LIN {X 0,Y 44.352,Z 475.064,A -85,B 0,C 180,E1 -30779.969,E2 -30779.969} C_VEL
LIN {X 0,Y 35.444,Z 475.32,A -85,B 0,C 180,E1 -30787.589,E2 -30787.589} C_VEL
LIN {X 0,Y 29.276,Z 474.961,A -85,B 0,C 180,E1 -30796.255,E2 -30796.255} C_VEL
LIN {X 0,Y 22.466,Z 473.712,A -85,B 0,C 180,E1 -30814.655,E2 -30814.655} C_VEL
LIN {X 0,Y 19.51,Z 472.671,A -85,B 0,C 180,E1 -30828.383,E2 -30828.383} C_VEL
LIN {X 0,Y 17,Z 471.328,A -85,B 0,C 180,E1 -30844.896,E2 -30844.896} C_VEL
LIN {X 0,Y 16.61,Z 467.855,A -85,B 0,C 180,E1 -30884.85,E2 -30884.85} C_VEL
LIN {X 0,Y 19.552,Z 465.667,A -85,B 0,C 180,E1 -30899.911,E2 -30899.911} C_VEL
LIN {X 0,Y 20.907,Z 464.867,A -85,B 0,C 180,E1 -30903.377,E2 -30903.377} C_VEL
LIN {X 0,Y 31.045,Z 458.924,A -85,B 0,C 180,E1 -30917.285,E2 -30917.285} C_VEL
LIN {X 0,Y 41.244,Z 451.859,A -85,B 0,C 180,E1 -30924.051,E2 -30924.051} C_VEL
LIN {X 0,Y 51.399,Z 443.285,A -85,B 0,C 180,E1 -30928.242,E2 -30928.242} C_VEL
LIN {X 0,Y 60.425,Z 433.954,A -85,B 0,C 180,E1 -30930.74,E2 -30930.74} C_VEL
LIN {X 0,Y 68.419,Z 423.904,A -85,B 0,C 180,E1 -30932.379,E2 -30932.379} C_VEL
LIN {X 0,Y 75.556,Z 412.822,A -85,B 0,C 180,E1 -30933.554,E2 -30933.554} C_VEL
LIN {X 0,Y 81.798,Z 400.333,A -85,B 0,C 180,E1 -30934.484,E2 -30934.484} C_VEL
LIN {X 0,Y 86.455,Z 387.975,A -85,B 0,C 180,E1 -30935.15,E2 -30935.15} C_VEL
LIN {X 0,Y 89.843,Z 375.107,A -85,B 0,C 180,E1 -30935.553,E2 -30935.553} C_VEL
LIN {X 0,Y 91.232,Z 367.157,A -85,B 0,C 180,E1 -30935.77,E2 -30935.77} C_VEL
LIN {X 0,Y 90.551,Z 364.005,A -85,B 0,C 180,E1 -30939.811,E2 -30939.811} C_VEL
LIN {X 0,Y 90.135,Z 362.029,A -85,B 0,C 180,E1 -30943.737,E2 -30943.737} C_VEL
LIN {X 0,Y 90.077,Z 360.543,A -85,B 0,C 180,E1 -30949.224,E2 -30949.224} C_VEL
LIN {X 0,Y 90.153,Z 360.685,A -85,B 0,C 180,E1 -30951.42,E2 -30951.42} C_VEL
LIN {X 0,Y 90.382,Z 362.249,A -85,B 0,C 180,E1 -30954.99,E2 -30954.99} C_VEL
LIN {X 0,Y 91.055,Z 365.77,A -85,B 0,C 180,E1 -30959.767,E2 -30959.767} C_VEL
LIN {X 0,Y 91.295,Z 367.107,A -85,B 0,C 180,E1 -30961.202,E2 -30961.202} C_VEL
LIN {X 0,Y 89.068,Z 378.985,A -85,B 0,C 180,E1 -30961.537,E2 -30961.537} C_VEL
LIN {X 0,Y 85.544,Z 391.077,A -85,B 0,C 180,E1 -30961.898,E2 -30961.898} C_VEL
LIN {X 0,Y 80.897,Z 402.684,A -85,B 0,C 180,E1 -30962.384,E2 -30962.384} C_VEL
LIN {X 0,Y 74.797,Z 414.427,A -85,B 0,C 180,E1 -30963.235,E2 -30963.235} C_VEL
LIN {X 0,Y 67.835,Z 424.975,A -85,B 0,C 180,E1 -30964.236,E2 -30964.236} C_VEL
LIN {X 0,Y 60.062,Z 434.695,A -85,B 0,C 180,E1 -30965.908,E2 -30965.908} C_VEL
LIN {X 0,Y 51.56,Z 443.447,A -85,B 0,C 180,E1 -30968.156,E2 -30968.156} C_VEL
LIN {X 0,Y 43.026,Z 450.805,A -85,B 0,C 180,E1 -30971.424,E2 -30971.424} C_VEL
LIN {X 0,Y 33.141,Z 457.934,A -85,B 0,C 180,E1 -30977.361,E2 -30977.361} C_VEL
LIN {X 0,Y 23.824,Z 463.593,A -85,B 0,C 180,E1 -30987.718,E2 -30987.718} C_VEL
LIN {X 0,Y 16.117,Z 468.031,A -85,B 0,C 180,E1 -31009.123,E2 -31009.123} C_VEL
LIN {X 0,Y 12.856,Z 471.354,A -85,B 0,C 180,E1 -31049.974,E2 -31049.974} C_VEL
LIN {X 0,Y 14.333,Z 472.961,A -85,B 0,C 180,E1 -31079.335,E2 -31079.335} C_VEL
LIN {X 0,Y 18.445,Z 474.174,A -85,B 0,C 180,E1 -31099.618,E2 -31099.618} C_VEL
LIN {X 0,Y 30.007,Z 475.461,A -85,B 0,C 180,E1 -31119.494,E2 -31119.494} C_VEL
LIN {X 0,Y 43.171,Z 475.216,A -85,B 0,C 180,E1 -31127.587,E2 -31127.587} C_VEL
LIN {X 0,Y 45.42,Z 475.038,A -85,B 0,C 180,E1 -31129.643,E2 -31129.643} C_VEL
LIN {X 0,Y 35.285,Z 475.456,A -85,B 0,C 180,E1 -31134.698,E2 -31134.698} C_VEL
LIN {X 0,Y 28.108,Z 475.182,A -85,B 0,C 180,E1 -31140.611,E2 -31140.611} C_VEL
LIN {X 0,Y 16.727,Z 473.532,A -85,B 0,C 180,E1 -31162.379,E2 -31162.379} C_VEL
LIN {X 0,Y 12.169,Z 470.625,A -85,B 0,C 180,E1 -31213.245,E2 -31213.245} C_VEL
LIN {X 0,Y 17.378,Z 466.834,A -85,B 0,C 180,E1 -31253.876,E2 -31253.876} C_VEL
LIN {X 0,Y 20.907,Z 464.867,A -85,B 0,C 180,E1 -31263.377,E2 -31263.377} C_VEL
LIN {X 0,Y 24.929,Z 462.408,A -85,B 0,C 180,E1 -31272.173,E2 -31272.173} C_VEL
LIN {X 0,Y 31.341,Z 457.783,A -85,B 0,C 180,E1 -31284.487,E2 -31284.487} C_VEL
LIN {X 0,Y 36.841,Z 453.625,A -85,B 0,C 180,E1 -31291.319,E2 -31291.319} C_VEL
LIN {X 0,Y 41.286,Z 450.18,A -85,B 0,C 180,E1 -31294.2,E2 -31294.2} C_VEL
LIN {X 0,Y 42.822,Z 448.958,A -85,B 0,C 180,E1 -31294.69,E2 -31294.69} C_VEL
LIN {X 0,Y 52.866,Z 440.168,A -85,B 0,C 180,E1 -31296.525,E2 -31296.525} C_VEL
LIN {X 0,Y 61.715,Z 430.571,A -85,B 0,C 180,E1 -31297.721,E2 -31297.721} C_VEL
LIN {X 0,Y 69.846,Z 419.682,A -85,B 0,C 180,E1 -31298.564,E2 -31298.564} C_VEL
LIN {X 0,Y 76.76,Z 408.103,A -85,B 0,C 180,E1 -31299.08,E2 -31299.08} C_VEL
LIN {X 0,Y 82.489,Z 395.479,A -85,B 0,C 180,E1 -31299.596,E2 -31299.596} C_VEL
LIN {X 0,Y 86.894,Z 382.266,A -85,B 0,C 180,E1 -31299.901,E2 -31299.901} C_VEL
LIN {X 0,Y 89.352,Z 371.228,A -85,B 0,C 180,E1 -31300.213,E2 -31300.213} C_VEL
LIN {X 0,Y 89.079,Z 369.034,A -85,B 0,C 180,E1 -31304.174,E2 -31304.174} C_VEL
LIN {X 0,Y 89.081,Z 367.713,A -85,B 0,C 180,E1 -31309.102,E2 -31309.102} C_VEL
LIN {X 0,Y 89.155,Z 367.905,A -85,B 0,C 180,E1 -31311.516,E2 -31311.516} C_VEL
LIN {X 0,Y 89.285,Z 369.744,A -85,B 0,C 180,E1 -31314.932,E2 -31314.932} C_VEL
LIN {X 0,Y 89.423,Z 371.225,A -85,B 0,C 180,E1 -31316.847,E2 -31316.847} C_VEL
LIN {X 0,Y 86.648,Z 383.385,A -85,B 0,C 180,E1 -31317.049,E2 -31317.049} C_VEL
LIN {X 0,Y 82.237,Z 396.373,A -85,B 0,C 180,E1 -31317.29,E2 -31317.29} C_VEL
LIN {X 0,Y 76.501,Z 408.793,A -85,B 0,C 180,E1 -31317.622,E2 -31317.622} C_VEL
LIN {X 0,Y 69.444,Z 420.477,A -85,B 0,C 180,E1 -31318.11,E2 -31318.11} C_VEL
LIN {X 0,Y 61.512,Z 431.021,A -85,B 0,C 180,E1 -31318.884,E2 -31318.884} C_VEL
LIN {X 0,Y 51.948,Z 441.238,A -85,B 0,C 180,E1 -31320.159,E2 -31320.159} C_VEL
LIN {X 0,Y 42.197,Z 449.644,A -85,B 0,C 180,E1 -31321.906,E2 -31321.906} C_VEL
LIN {X 0,Y 31.753,Z 456.992,A -85,B 0,C 180,E1 -31325.014,E2 -31325.014} C_VEL
LIN {X 0,Y 21.457,Z 462.846,A -85,B 0,C 180,E1 -31330.621,E2 -31330.621} C_VEL
LIN {X 0,Y 11.705,Z 467.437,A -85,B 0,C 180,E1 -31345.693,E2 -31345.693} C_VEL
LIN {X 0,Y 5.755,Z 470.89,A -85,B 0,C 180,E1 -31409.942,E2 -31409.942} C_VEL
LIN {X 0,Y 8.864,Z 472.578,A -85,B 0,C 180,E1 -31462.389,E2 -31462.389} C_VEL
LIN {X 0,Y 14.856,Z 473.854,A -85,B 0,C 180,E1 -31481.038,E2 -31481.038} C_VEL
LIN {X 0,Y 18.473,Z 474.395,A -85,B 0,C 180,E1 -31491.228,E2 -31491.228} C_VEL
LIN {X 0,Y 7.422,Z 472.126,A -85,B 0,C 180,E1 -31518.903,E2 -31518.903} C_VEL
LIN {X 0,Y 7.924,Z 468.795,A -85,B 0,C 180,E1 -31617.88,E2 -31617.88} C_VEL
LIN {X 0,Y 17.76,Z 464.463,A -85,B 0,C 180,E1 -31642.35,E2 -31642.35} C_VEL
LIN {X 0,Y 27.823,Z 459.169,A -85,B 0,C 180,E1 -31649.714,E2 -31649.714} C_VEL
LIN {X 0,Y 39.187,Z 451.742,A -85,B 0,C 180,E1 -31653.749,E2 -31653.749} C_VEL
LIN {X 0,Y 42.822,Z 448.958,A -85,B 0,C 180,E1 -31654.69,E2 -31654.69} C_VEL
LIN {X 0,Y 47.201,Z 445.25,A -85,B 0,C 180,E1 -31656.437,E2 -31656.437} C_VEL
LIN {X 0,Y 53.768,Z 438.706,A -85,B 0,C 180,E1 -31660.493,E2 -31660.493} C_VEL
LIN {X 0,Y 60.023,Z 431.698,A -85,B 0,C 180,E1 -31663.652,E2 -31663.652} C_VEL
LIN {X 0,Y 63.737,Z 427.099,A -85,B 0,C 180,E1 -31664.312,E2 -31664.312} C_VEL
LIN {X 0,Y 71.17,Z 416.473,A -85,B 0,C 180,E1 -31664.339,E2 -31664.339} C_VEL
LIN {X 0,Y 77.412,Z 405.321,A -85,B 0,C 180,E1 -31664.408,E2 -31664.408} C_VEL
LIN {X 0,Y 82.253,Z 394.264,A -85,B 0,C 180,E1 -31664.533,E2 -31664.533} C_VEL
LIN {X 0,Y 86.454,Z 381.246,A -85,B 0,C 180,E1 -31664.574,E2 -31664.574} C_VEL
LIN {X 0,Y 87.7,Z 376.105,A -85,B 0,C 180,E1 -31664.651,E2 -31664.651} C_VEL
LIN {X 0,Y 87.796,Z 374.873,A -85,B 0,C 180,E1 -31668.94,E2 -31668.94} C_VEL
LIN {X 0,Y 87.87,Z 374.888,A -85,B 0,C 180,E1 -31671.103,E2 -31671.103} C_VEL
LIN {X 0,Y 87.82,Z 375.621,A -85,B 0,C 180,E1 -31672.324,E2 -31672.324} C_VEL
LIN {X 0,Y 84.682,Z 387.47,A -85,B 0,C 180,E1 -31672.317,E2 -31672.317} C_VEL
LIN {X 0,Y 80.762,Z 398.126,A -85,B 0,C 180,E1 -31672.316,E2 -31672.316} C_VEL
LIN {X 0,Y 75.353,Z 409.407,A -85,B 0,C 180,E1 -31672.325,E2 -31672.325} C_VEL
LIN {X 0,Y 68.277,Z 420.941,A -85,B 0,C 180,E1 -31672.229,E2 -31672.229} C_VEL
LIN {X 0,Y 60.29,Z 431.399,A -85,B 0,C 180,E1 -31672.28,E2 -31672.28} C_VEL
LIN {X 0,Y 51.566,Z 440.648,A -85,B 0,C 180,E1 -31672.329,E2 -31672.329} C_VEL
LIN {X 0,Y 42.559,Z 448.483,A -85,B 0,C 180,E1 -31672.28,E2 -31672.28} C_VEL
LIN {X 0,Y 31.928,Z 456.018,A -85,B 0,C 180,E1 -31672.185,E2 -31672.185} C_VEL
LIN {X 0,Y 21.33,Z 462.036,A -85,B 0,C 180,E1 -31671.398,E2 -31671.398} C_VEL
LIN {X 0,Y 14.261,Z 465.357,A -85,B 0,C 180,E1 -31670.415,E2 -31670.415} C_VEL
LIN {X 0,Y 14.451,Z 465.266,A -85,B 0,C 180,E1 -31666.668,E2 -31666.668} C_VEL
LIN {X 0,Y 26.23,Z 459.394,A -85,B 0,C 180,E1 -31664.513,E2 -31664.513} C_VEL
LIN {X 0,Y 38.36,Z 451.621,A -85,B 0,C 180,E1 -31664.154,E2 -31664.154} C_VEL
LIN {X 0,Y 47.477,Z 444.337,A -85,B 0,C 180,E1 -31664.217,E2 -31664.217} C_VEL
LIN {X 0,Y 56.635,Z 435.43,A -85,B 0,C 180,E1 -31664.282,E2 -31664.282} C_VEL
LIN {X 0,Y 63.737,Z 427.099,A -85,B 0,C 180,E1 -31664.312,E2 -31664.312} C_VEL
LIN {X 0,Y 67.306,Z 428.339,A -85,B 0,C 180,E1 -31664.345,E2 -31664.345} C_VEL
LIN {X 0,Y 67.306,Z 600,A -85,B 0,C 180,E1 -31664.345,E2 -31664.345} C_VEL
LIN {X 0,Y 67.306,Z 600,A -85,B 0,C 180,E1 -31664.345,E2 -31664.345}

QRS_NEXT_CUT()

QRS_NEXT()
QRS_HOME()

END
